FUNCTION_BLOCK Gate Implements itfAutoManual
VAR_INPUT
	GateInput : GateI;
END_VAR
VAR_OUTPUT
	GateOutput : GateO;
END_VAR
VAR
Actuate : itfActuate;
ActuateComp : itfActuateImplement;	

END_VAR

Map();

METHOD PRIVATE Map : BOOL
VAR_INPUT
END_VAR
Actuate := ActuateComp;

Actuate.pStart := GateInput.Open;
Actuate.pStop := GateInput.Close;
GateOutput.Coil := Actuate.pCoil;
END_METHOD

{warning 'add method implementation '}
METHOD mAutoOff : BOOL
Actuate.mTurnOffAuto();
END_METHOD

{warning 'add method implementation '}
METHOD mAutoOn : BOOL
Actuate.mTurnOnAuto();
END_METHOD

{warning 'add method implementation '}
METHOD mFault : BOOL
END_METHOD

{warning 'add method implementation '}
METHOD mManual : BOOL
Actuate.mTurnOnManual();
Actuate.mTurnOffManual();
END_METHOD

{warning 'add method implementation '}
METHOD mRunning : BOOL
mRunning := Actuate.pCoil;
END_METHOD

END_FUNCTION_BLOCK

(* stored: Version 1.1.0.1, ProductVersion 3.1.4024.12
   POU Gate: Id {704da9fa-6781-4768-a110-21002bb7eecc}, SpecialFunc None
   Method Map: Id {64ffc566-33e0-413c-9a01-caec3ef8c01d}
   Method mAutoOff: Id {4903f606-3d6d-4c13-b763-581cb21c69f2}
   Method mAutoOn: Id {eeef2779-bbe0-4491-9ad7-6f146cc323cf}
   Method mFault: Id {8cf7b193-0bc2-4f0e-8197-f4b484b71478}
   Method mManual: Id {d447e9aa-eac8-4621-bd60-518199c8c6be}
   Method mRunning: Id {e78dcd01-4b36-4027-8107-7a6c22109049} *)
